// TIA Portal V20 export
// export: Created 2026-04-11T06:02:30.5867448Z, ExportSetting WithDefaults, DisplayName Totally Integrated Automation Portal, DisplayVersion V20, DisplayName TIA Portal Openness, DisplayVersion V20, DisplayName TIA Portal Version Control Interface, DisplayVersion V20, DisplayName STEP 7 Professional, DisplayVersion V20, DisplayName STEP 7 Safety, DisplayVersion V20, DisplayName WinCC Basic/Comfort/Advanced, DisplayVersion V20, DisplayName WinCC Unified, DisplayVersion V20
TYPE "udtHMI_Brabender_Output"
// stored: IsFailsafeCompliant false
   STRUCT
      iFunction { S7_SetPoint := 'True'} : Int;   // Function codes (see manual or FB comments)
      iOperatingMode { S7_SetPoint := 'True'} : Int;   // Operating modes (see manual or FB comments)
      rDecadeSwitch { S7_SetPoint := 'True'} : Real;   // Decade switch
      rSetpoint { S7_SetPoint := 'True'} : Real;   // Setpoint [kg/h]
      rSetpointAnalog { S7_SetPoint := 'True'} : Real;   // Setpoint [%] for analogue control
      rSetpointCleaning { S7_SetPoint := 'True'} : Real;   // Setpoint [%] for DI/cleaning
      rControlDifference { S7_SetPoint := 'True'} : Real;   // Control difference [%]
      rBulkDensity { S7_SetPoint := 'True'} : Real;   // Bulk density [kg/l]
      rCheckMaxOutput { S7_SetPoint := 'True'} : Real;   // Check. max. output [kg/hr]
      rPTermController { S7_SetPoint := 'True'} : Real;   // P-term controller
      rITermController { S7_SetPoint := 'True'} : Real;   // I-term controller
      rActualDTermController { S7_SetPoint := 'True'} : Real;   // D-term controller
      rControllerAdaptation { S7_SetPoint := 'True'} : Real;   // Controller adaptation
      rActualFillLevelMin { S7_SetPoint := 'True'} : Real;   // Filling level minimum [%]
      rActualFillLevelMax { S7_SetPoint := 'True'} : Real;   // Filling level maximum [%]
   END_STRUCT;
END_TYPE
